// TwinCAT 3 PLC project PLCproject1
// ProgramVersion: 3.1.4023.0
// libraries:
//   Tc2_Standard, * (Beckhoff Automation GmbH)
//   Tc2_System, * (Beckhoff Automation GmbH)
//   Tc2_Utilities, * (Beckhoff Automation GmbH)
//   Tc3_Module, * (Beckhoff Automation GmbH)
// project tree:
//   01_InfeedConveyor/ InfeedConveyor.TcGVL (not stored)
//   02_PickandPlace/ PickAndPlace.TcGVL (not stored), PickAndPlace_Pick.TcDUT (not stored)
//   GVLs/ PersistentExample.TcGVL (not stored)
//   / PlcTask.TcTTO
//   POUs/ MAIN.TcPOU, SavePersistentVariables.TcPOU (not stored)

CONFIGURATION PLCproject1
    RESOURCE PLC ON TwinCAT3
        TASK PlcTask(INTERVAL := T#10ms, PRIORITY := 20);
        PROGRAM MAIN WITH PlcTask : MAIN;
    END_RESOURCE
END_CONFIGURATION

// ---- POUs/MAIN.TcPOU
PROGRAM MAIN 
VAR
END_VAR

SavePersistentVariables ();

END_PROGRAM
